RoboDK station: Proyecto_RoboDK_PR2 1.rdk

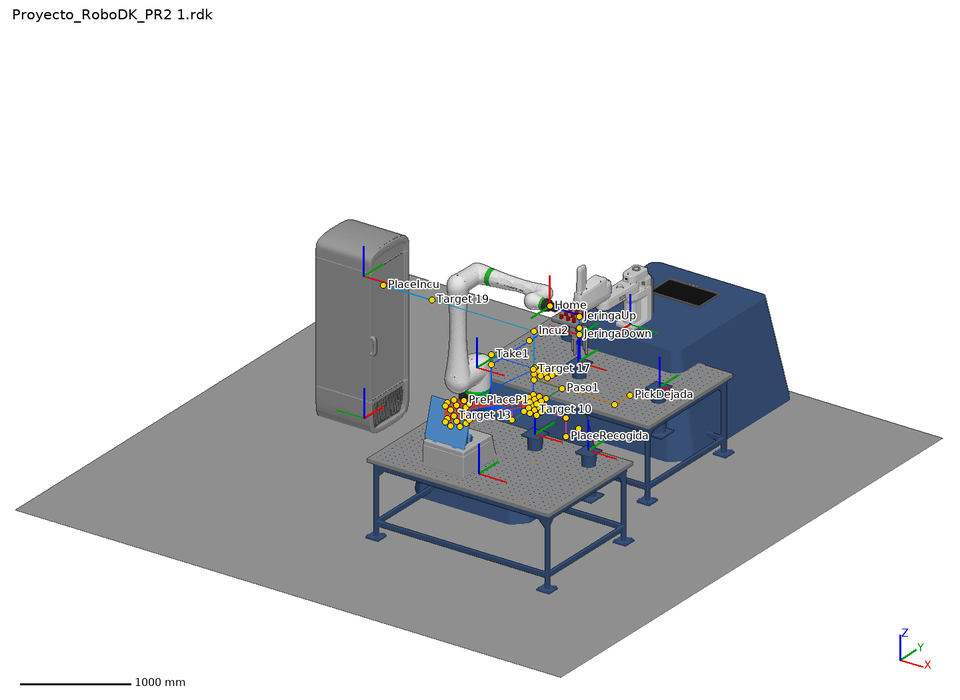
[picture v0: the station drawn from its stored meshes, robots at their saved joint values, targets as dots, program paths as lines]
Station pRUEBA (saved by RoboDK 5.9.4). Poses are relative to the parent item; angles as X-Y-Z fixed-axis rotations.
  - frame Frame 1 at (0, 0, 0) mm
    - object Floor at (-1500, 1500, 0) mm, size 3000 x 3000 x 0 mm, geometry from Floor.sld
    - object Floor at (1500, -1500, 0) mm, size 3000 x 3000 x 0 mm, geometry from Floor.sld
    - object Floor at (1500, 1500, 0) mm, size 3000 x 3000 x 0 mm, geometry from Floor.sld
    - object Floor at (-1500, -1500, 0) mm, size 3000 x 3000 x 0 mm, geometry from Floor.sld
    - object Table 2000x1200x800mm at (300, -1000, 800) mm, size 2020 x 1340 x 800 mm, geometry from Table-2000x1200x800mm.sld
    - object Table 2000x1200x800mm at (0, 1000, 800) mm, size 2020 x 1340 x 800 mm, geometry from Table-2000x1200x800mm.sld
    - object Pedestal H750mm (Type 2) at (320, 0, 0) mm, size 1266.8 x 1400.5 x 750 mm, geometry from Pedestal-H750mm-Type-2.sld
    - object Pedestal H1000mm (Type 2) at (580, 2100, 0) mm, size 1689.1 x 1867.3 x 1000 mm, geometry from Pedestal-H1000mm-Type-2.sld
    - object Pedestal H36in (Type 1) at (1400, 40, -20) mm, size 200 x 200 x 457.2 mm, geometry from Pedestal-H36in-Type-1.sld
    - object Pedestal H36in (Type 1) at (530, 40, -20) mm, size 200 x 200 x 457.2 mm, geometry from Pedestal-H36in-Type-1.sld
    - object Pedestal H36in (Type 1) at (1050, -1400, -10) mm, size 200 x 200 x 457.2 mm, geometry from Pedestal-H36in-Type-1.sld
    - object Pedestal H36in (Type 1) at (1640, -1400, -20) mm, size 200 x 200 x 457.2 mm, geometry from Pedestal-H36in-Type-1.sld
    - object Centrifugadora at (440, -1500, 800) mm, size 484.9 x 550 x 655.5 mm, geometry from Centrifugadora.stl
    - object Display Panel 24in at (590, 2390, 1010) mm, rotated rx 0 ry -90 rz 90 deg, size 43 x 556.4 x 342.2 mm, geometry from Display-Panel-24in.sld
  - frame Adept Cobra s800 Base at (530, 1620, 1000) mm, rotated rx 0 ry 0 rz -90 deg
    - robot myScara (model Adept Cobra s800): 4 axes, payload 2 kg, reach 800 mm, repeatability 0.018 mm, weight 43 kg
        modified DH rows (alpha deg, a mm, theta deg, d mm): 0, 0, 0, 0; 0, 425, 0, 0; 0, 375, 0, 184 linear; 180, 0, 0, 0
        joint limits [-105, -157.5, 0, -360] to [105, 157.5, 210, 360]; home [0, 0, 0, 0]; saved at [0, 0, 30, 90]
      - frame FrameScaraTool at (0, 0, 0) mm
        - object ScaraTool at (0, 0, 0) mm, size 193.5 x 193.5 x 277.1 mm, geometry from robodk.stl
    - target JeringaUp (Cartesian target) at (800, 0, 394) mm, rotated rx 180 ry 0 rz 0 deg; joints [0, 0, 210, 0] of myScara
    - target JeringaPreDown (Cartesian target) at (800, 0, 284) mm, rotated rx 180 ry 0 rz 0 deg; joints [0, 0, 100, 0, 0, 0] of myScara
    - target JeringaDown (Cartesian target) at (800, 0, 214) mm, rotated rx 180 ry 0 rz 0 deg; joints [0, 0, 30, 0, 0, 0] of myScara
    - target Sustancia2 (Cartesian target) at (800, 0, 214) mm, rotated rx 180 ry 0 rz -90 deg; joints [0, 0, 30, 90, 0, 0] of myScara
    - target Sustancia3 (Cartesian target) at (800, 0, 214) mm, rotated rx -180 ry 0 rz -180 deg; joints [0, 0, 30, 180, 0, 0] of myScara
    - target Alchol (Cartesian target) at (800, 0, 214) mm, rotated rx -180 ry 0 rz 90 deg; joints [0, 0, 30, 270, 0, 0] of myScara
    - target PreSustancia2 (Cartesian target) at (800, 0, 284) mm, rotated rx 180 ry 0 rz -90 deg; joints [0, 0, 100, 90] of myScara
    - target PreSustancia3 (Cartesian target) at (800, 0, 284) mm, rotated rx -180 ry 0 rz -180 deg; joints [0, 0, 100, 180] of myScara
    - target PreAlchol (Cartesian target) at (800, 0, 284) mm, rotated rx -180 ry 0 rz 90 deg; joints [0, 0, 100, 270] of myScara
    - target Target 10 (Cartesian target) at (2240, 517.5, 180) mm, rotated rx 180 ry 0 rz 90 deg; joints [143.001, -36.832, -136.065, 0, 46.065, -143.001] of myRobotUR
    - target Target 11 (Cartesian target) at (2170, 517.5, 180) mm, rotated rx 180 ry 0 rz 90 deg; joints [145.986, -35.485, -134.651, 0, 44.651, -145.986] of myRobotUR
    - target Target 12 (Cartesian target) at (2170, 590, 180) mm, rotated rx -180 ry 0 rz 90 deg; joints [148.02, -38.44, -137.769, 0, 47.769, -148.02] of myRobotUR
    - target Target 13 (Cartesian target) at (2840, 50, 230) mm, rotated rx 180 ry 0 rz 90 deg; joints [106.738, -40.272, -144.565, 0, 54.565, -106.738] of myRobotUR
    - target Target 14 (Cartesian target) at (2240, 590, 180) mm, rotated rx -180 ry 0 rz 90 deg; joints [145.135, -39.762, -139.179, 0, 49.179, -145.135] of myRobotUR
    - target Target 15 (Cartesian target) at (2315, 590, 180) mm, rotated rx 180 ry 0 rz 90 deg; joints [142.232, -41.383, -140.921, 0, 50.921, -142.232] of myRobotUR
    - target Target 16 (Cartesian target) at (2315, 590, 180) mm, rotated rx 180 ry 0 rz 90 deg; joints [142.232, -41.383, -140.921, 0, 50.921, -142.232] of myRobotUR
    - target Target 17 (Cartesian target) at (2170, 450, 540) mm, rotated rx 180 ry 0 rz 90 deg; joints [143.864, -20.056, -157.055, 0, 67.055, -143.864] of myRobotUR
    - target Target 18 (Cartesian target) at (1795, 200, -45) mm, rotated rx 0 ry -90 rz -90 deg; joints [12.327, 57.498, -112.698, -13.327, 112.147, -5.103] of myRobotUR
    - target Target 19 (Cartesian target) at (1355, -1230, 440) mm, rotated rx 0 ry -90 rz 90 deg; joints [162.189, 12.692, -58.671, 20.612, 60.328, -10.547] of myRobotUR
    - target Target 20 (Cartesian target) at (2140, 200, -50) mm, rotated rx 0 ry -90 rz -90 deg; joints [-25.299, 52.835, -105.784, 26.16, 104.237, 6.888] of myRobotUR
    - target Target 21 (Cartesian target) at (1120, -100, -45) mm, rotated rx 0 ry -90 rz 0 deg; joints [64.725, 54.326, -114.186, 27.366, 111.745, 10.855] of myRobotUR
    - target Target 22 (Cartesian target) at (800, 0, 214) mm, rotated rx 180 ry 0 rz 0 deg; joints [72.717, 31.504, -45.613, 0, -44.387, -162.717] of myRobotUR
    - target Target 23 (Cartesian target) at (1905, 450, 1070) mm, rotated rx 0 ry -90 rz -90 deg; joints [0, 0, 0, 0, 0, 0] of myRobotUR
  - frame Fanuc CRX-25iA Base at (50, -100, 1120) mm
    - robot myRobotUR (model Fanuc CRX-25iA): 6 axes, payload 25 kg, reach 1889 mm, repeatability 0.05 mm, weight 135 kg
        modified DH rows (alpha deg, a mm, theta deg, d mm): 0, 0, 0, 370; -90, 0, -90, 0; 0, 950, 0, 0; -90, 0, 0, 750; 90, 0, 0, -185; -90, 0, 0, 180
        base shift (0, 0, -370) mm
        joint limits [-180, -180, -270, -190, -180, -225] to [180, 180, 270, 190, 180, 225]; home [0, 0, 0, 0, 0, 0]; saved at [0, 0, 0, 0, 0, 0]
      - frame RobotiQ 2F-140 Gripper (Mechanism) Base at (0, 0, 0) mm
        - robot RobotiQ 2F-140 Gripper (Mechanism) (model RobotiQ 2F140): 1 axes, payload 5 kg
            joint limits [0] to [140]; home [140]; saved at [40]
          - tool Tool 1, TCP at (0, 0, 200) mm
            - object Soporte1 at (-20, 30, 45) mm, rotated rx 90 ry 0 rz 90 deg, size 266.4 x 266.4 x 36 mm, geometry from soporteprobeta.stl
              - object P1 at (5, 0, 0) mm, size 36.4 x 36.5 x 72.9 mm, geometry from probeta.stl
              - object P2 at (75, 0, 0) mm, size 36.4 x 36.5 x 72.9 mm, geometry from probeta.stl
              - object P3 at (150, 0, 0) mm, size 36.4 x 36.5 x 72.9 mm, geometry from probeta.stl
              - object P4 at (150, 72.5, 0) mm, size 36.4 x 36.5 x 72.9 mm, geometry from probeta.stl
              - object P5 at (75, 72.5, 0) mm, size 36.4 x 36.5 x 72.9 mm, geometry from probeta.stl
              - object P6 at (5, 72.5, 0) mm, size 36.4 x 36.5 x 72.9 mm, geometry from probeta.stl
              - object P7 at (5, 145, 0) mm, size 36.4 x 36.5 x 72.9 mm, geometry from probeta.stl
              - object P8 at (75, 145, 0) mm, size 36.4 x 36.5 x 72.9 mm, geometry from probeta.stl
              - object P9 at (150, 145, 0) mm, size 36.4 x 36.5 x 72.9 mm, geometry from probeta.stl
        - target GarraOpen (Cartesian target) at (0, 0, 0) mm; joints [140, 0, 0, 0, 0, 0] of RobotiQ 2F-140 Gripper (Mechanism)
        - target GarraPick (Cartesian target) at (0, 0, 0) mm; joints [40, 0, 30, 270] of RobotiQ 2F-140 Gripper (Mechanism)
  - frame IncubadoraMECA at (-1500, 340, 0) mm, rotated rx 0 ry 0 rz 90 deg
    - robot Refrigeradora: 1 axes
        modified DH rows (alpha deg, a mm, theta deg, d mm): 0, 0, 0, 0 linear
        base shift (0, 0, 0) mm, rotated rx 0 ry 90 rz 0 deg
        joint limits [0] to [600]; home [0]; saved at [0]
    - target DoorClose (Cartesian target) at (0, 0, 0) mm; joints [0, 54.489, -114.295, 25.89, 112.102, 10.349] of Refrigeradora
    - target DoorOpen (Cartesian target) at (600, 0, 0) mm; joints [600, 54.489, -114.295, 25.89, 112.102, 10.349] of Refrigeradora
  - frame Dejada at (1410, 820, 940) mm
    - target PickDejada (Cartesian target) at (-100, -315, 15) mm, rotated rx 0 ry -90 rz -90 deg; joints [21.278, 62.791, -64.214, 70.676, 80.917, -24.237] of myRobotUR
    - target PrePickDejada (Cartesian target) at (-100, -555, 15) mm, rotated rx 0 ry -90 rz -90 deg; joints [9.654, 60.648, -68.477, 81.008, 86.473, -21.245] of myRobotUR
    - target Home (Cartesian target) at (-430, -1105, 1130) mm, rotated rx 0 ry -90 rz -180 deg; joints [0, 0, 0, 0, 0, 0] of myRobotUR
  - frame Pinchazo at (520, 820, 940) mm
    - target PlacePinchazo/Pin2 (Cartesian target) at (-90, -320, 15) mm, rotated rx 0 ry -90 rz -90 deg; joints [64.725, 54.326, -114.186, 27.366, 111.745, 10.855] of myRobotUR
    - target PrePlacePinchazo (Cartesian target) at (-100, -555, 15) mm, rotated rx 0 ry -90 rz -90 deg; joints [39.607, 59.804, -135.062, 59.694, 116.826, 37.672] of myRobotUR
    - target Pin1 (Cartesian target) at (-20, -320, 15) mm, rotated rx 0 ry -90 rz -90 deg; joints [57.411, 52.743, -110.092, 34.243, 106.825, 11.146] of myRobotUR
    - target Pin3 (Cartesian target) at (-170, -320, 15) mm, rotated rx 0 ry -90 rz -90 deg; joints [74.441, 56.789, -118.585, 17.593, 117.447, 8.315] of myRobotUR
    - target Pin4 (Cartesian target) at (-170, -390, 15) mm, rotated rx 0 ry -90 rz -90 deg; joints [71.034, 59.762, -126.932, 23.265, 124.628, 13.729] of myRobotUR
    - target Pin5 (Cartesian target) at (-90, -390, 15) mm, rotated rx 0 ry -90 rz -90 deg; joints [59.932, 55.868, -120.613, 33.929, 116.149, 16.513] of myRobotUR
    - target Pin6 (Cartesian target) at (-20, -390, 15) mm, rotated rx 0 ry -90 rz -90 deg; joints [52.114, 53.534, -115.301, 40.717, 109.712, 16.188] of myRobotUR
    - target Pin7 (Cartesian target) at (-20, -460, 15) mm, rotated rx 0 ry -90 rz -90 deg; joints [45.12, 54.354, -120.163, 49.035, 110.857, 22.297] of myRobotUR
    - target Pin8 (Cartesian target) at (-90, -460, 15) mm, rotated rx 0 ry -90 rz -90 deg; joints [52.947, 57.441, -126.856, 43.337, 118.6, 24.308] of myRobotUR
    - target Pin9 (Cartesian target) at (-170, -460, 15) mm, rotated rx 0 ry -90 rz -90 deg; joints [65.053, 62.974, -135.774, 33.701, 130.522, 23.429] of myRobotUR
  - frame Incubadora at (-1500, 330, 1430) mm
    - target EncaraIncu (Cartesian target) at (1920, -65, -475) mm, rotated rx 0 ry -90 rz 0 deg; joints [18.17, 52.517, -103.492, 161.349, 77.192, 4.279] of myRobotUR
    - target Incu2 (Cartesian target) at (1920, -65, 10) mm, rotated rx 0 ry -90 rz 0 deg; joints [18.423, 11.864, -59.167, 158.797, 119.096, -10.683] of myRobotUR
    - target PlaceIncu (Cartesian target) at (260, -65, 10) mm, rotated rx 0 ry -90 rz 0 deg; joints [170.623, 35.683, -40.43, 14.285, 41.321, -10.826] of myRobotUR
    - target PrePlaceIncu (Cartesian target) at (800, -65, 10) mm, rotated rx 0 ry -90 rz 0 deg; joints [162.189, 12.692, -58.671, 20.612, 60.328, -10.547] of myRobotUR
  - frame Centrifugadora at (1050, -620, 940) mm
    - target Centri1 (Cartesian target) at (-550, 885, 500) mm, rotated rx 0 ry -90 rz 0 deg; joints [16.192, 15.174, -57.101, 160.923, 121.44, -10.226] of myRobotUR
    - target Centri2 (Cartesian target) at (-550, 700, 500) mm, rotated rx 0 ry -90 rz 0 deg; joints [-0.454, 11.696, -54.321, 180.559, 125.678, 0.326] of myRobotUR
    - target Centri3/Giro (Cartesian target) at (-550, 700, 500) mm, rotated rx 0 ry -90 rz -90 deg; joints [0, 0.179, -68.498, 90, 90, -21.502] of myRobotUR
    - target Centri4/Giro (Cartesian target) at (-550, 700, 500) mm, rotated rx 0 ry -90 rz -180 deg; joints [49.88, -8.528, -41.712, -60.721, 61.247, 40.627] of myRobotUR
    - target Centri5 (Cartesian target) at (-550, 100, 500) mm, rotated rx 0 ry -90 rz -180 deg; joints [-41.992, 3.157, -65.505, 44.688, 72.052, -16.952] of myRobotUR
    - target PrePlaceCentri (Cartesian target) at (-550, 100, 10) mm, rotated rx 0 ry -90 rz -180 deg; joints [136.977, -56.167, -55.961, -131.602, 114.156, 24.744] of myRobotUR
    - target PlaceCentri (Cartesian target) at (-320, 100, 10) mm, rotated rx 0 ry -90 rz -180 deg; joints [154.701, -52.835, -74.216, -153.84, 104.237, 6.888] of myRobotUR
    - target LlevarRecogida (Cartesian target) at (-320, 100, 200) mm, rotated rx 0 ry -90 rz -180 deg; joints [154.826, -35.816, -89.736, -154.826, 90.239, 0.112] of myRobotUR
    - target Paso1 (Cartesian target) at (-320, 885, 15) mm, rotated rx 0 ry -90 rz -90 deg; joints [20.272, 50.493, -105.389, 70.399, 95.275, 14.477] of myRobotUR
    - target Paso2 (Cartesian target) at (-320, 885, 15) mm, rotated rx 0 ry -90 rz -180 deg; joints [47.726, 52.078, -90.466, -47.727, 90.314, -0.345] of myRobotUR
    - target PrePaso3 (Cartesian target) at (-320, 445, 15) mm, rotated rx 0 ry -90 rz 180 deg; joints [12.327, 57.498, -112.698, -13.327, 112.147, -5.103] of myRobotUR
    - target Take1 (Cartesian target) at (-550, 100, 600) mm, rotated rx 0 ry -90 rz -180 deg; joints [136.75, 4.022, -125.669, -130.814, 64.868, -26.187] of myRobotUR
    - target Take2 (Cartesian target) at (-550, 100, 600) mm, rotated rx 180 ry 0 rz 0 deg; joints [119.485, 4.704, -152.458, 0, 62.458, -119.485] of myRobotUR
    - target Take3 (Cartesian target) at (-70, 100, 600) mm, rotated rx 180 ry 0 rz 0 deg; joints [145.25, -19.338, -156.721, 0, 66.721, -145.25] of myRobotUR
    - target Take4 (Cartesian target) at (-70, 70, 600) mm, rotated rx -180 ry 0 rz 0 deg; joints [143.864, -20.056, -157.055, 0, 67.055, -143.864] of myRobotUR
    - target PickP1 (Cartesian target) at (-70, 70, 240) mm, rotated rx 180 ry 0 rz 0 deg; joints [143.864, -32.854, -131.921, 0, 41.921, -143.864] of myRobotUR
    - target PrePickP1 (Cartesian target) at (-70, 70, 350) mm, rotated rx 180 ry 0 rz 0 deg; joints [143.864, -28.076, -139.387, 0, 49.387, -143.864] of myRobotUR
    - target PickP2 (Cartesian target) at (-70, 0, 240) mm, rotated rx 180 ry 0 rz 0 deg; joints [140.79, -34.237, -133.35, 0, 43.35, -140.79] of myRobotUR
    - target PrePickP2 (Cartesian target) at (-70, 0, 350) mm, rotated rx 180 ry 0 rz 0 deg; joints [140.79, -29.624, -140.622, 0, 50.622, -140.79] of myRobotUR
    - target PickP3 (Cartesian target) at (-70, -75, 240) mm, rotated rx -180 ry 0 rz 0 deg; joints [137.743, -35.912, -135.097, 0, 45.097, -137.743] of myRobotUR
    - target PrePickP3 (Cartesian target) at (-70, -75, 350) mm, rotated rx -180 ry 0 rz 0 deg; joints [137.743, -31.486, -142.156, 0, 52.156, -137.743] of myRobotUR
    - target PickP4 (Cartesian target) at (-2.5, -75, 240) mm, rotated rx -180 ry 0 rz 0 deg; joints [140.019, -38.472, -137.802, 0, 47.802, -140.019] of myRobotUR
    - target PrePickP4 (Cartesian target) at (-2.5, -75, 350) mm, rotated rx -180 ry 0 rz 0 deg; joints [140.019, -34.309, -144.577, 0, 54.577, -140.019] of myRobotUR
    - target PickP5 (Cartesian target) at (-2.5, 0, 240) mm, rotated rx 180 ry 0 rz 0 deg; joints [143.001, -36.832, -136.065, 0, 46.065, -143.001] of myRobotUR
    - target PrePickP5 (Cartesian target) at (-2.5, 0, 350) mm, rotated rx 180 ry 0 rz 0 deg; joints [143.001, -32.503, -143.016, 0, 53.016, -143.001] of myRobotUR
    - target PickP6 (Cartesian target) at (-2.5, 70, 240) mm, rotated rx 180 ry 0 rz 0 deg; joints [145.986, -35.485, -134.651, 0, 44.651, -145.986] of myRobotUR
    - target PrePickP6 (Cartesian target) at (-2.5, 70, 350) mm, rotated rx -180 ry 0 rz 0 deg; joints [145.986, -31.013, -141.762, 0, 51.762, -145.986] of myRobotUR
    - target PickP7 (Cartesian target) at (70, 70, 240) mm, rotated rx 180 ry 0 rz 0 deg; joints [148.02, -38.44, -137.769, 0, 47.769, -148.02] of myRobotUR
    - target PrePickP7 (Cartesian target) at (70, 70, 350) mm, rotated rx 180 ry 0 rz 0 deg; joints [148.02, -34.274, -144.546, 0, 54.546, -148.02] of myRobotUR
    - target PickP8 (Cartesian target) at (70, 0, 240) mm, rotated rx 180 ry 0 rz 0 deg; joints [145.135, -39.762, -139.179, 0, 49.179, -145.135] of myRobotUR
    - target PrePickP8 (Cartesian target) at (70, 0, 350) mm, rotated rx -180 ry 0 rz 0 deg; joints [145.135, -35.723, -145.828, 0, 55.828, -145.135] of myRobotUR
    - target PickP9 (Cartesian target) at (70, -75, 240) mm, rotated rx 180 ry 0 rz 0 deg; joints [142.232, -41.383, -140.921, 0, 50.921, -142.232] of myRobotUR
    - target PrePickP9 (Cartesian target) at (70, -75, 350) mm, rotated rx -180 ry 0 rz 0 deg; joints [142.232, -37.492, -147.428, 0, 57.428, -142.232] of myRobotUR
    - target PlaceP1 (Cartesian target) at (-390, -560, 290) mm, rotated rx -180 ry 0 rz 0 deg; joints [110.881, -40.337, -144.63, 0, 54.63, -110.881] of myRobotUR
    - target PrePlaceP1 (Cartesian target) at (-390, -560, 450) mm, rotated rx -180 ry 0 rz 0 deg; joints [110.881, -35.397, -154.371, 0, 64.371, -110.881] of myRobotUR
    - target PlaceP2 (Cartesian target) at (-290, -665, 290) mm, rotated rx 180 ry 0 rz 0 deg; joints [113.232, -47.852, -152.398, 0, 62.398, -113.232] of myRobotUR
    - target PrePlaceP2 (Cartesian target) at (-290, -665, 450) mm, rotated rx -180 ry 0 rz 0 deg; joints [113.232, -43.764, -161.652, 0, 71.652, -113.232] of myRobotUR
    - target PlaceP3 (Cartesian target) at (-380, -780, 290) mm, rotated rx -180 ry 0 rz 0 deg; joints [108.118, -51.381, -156.177, 0, 66.177, -108.118] of myRobotUR
    - target PrePlace3 (Cartesian target) at (-380, -780, 450) mm, rotated rx 180 ry 0 rz 0 deg; joints [108.118, -47.7, -165.375, 0, 75.375, -108.118] of myRobotUR
    - target PlaceP4 (Cartesian target) at (-490, -675, 290) mm, rotated rx 180 ry 0 rz 0 deg; joints [104.926, -43.35, -147.695, 0, 57.695, -104.926] of myRobotUR
    - target PrePlace4 (Cartesian target) at (-490, -675, 450) mm, rotated rx 180 ry 0 rz 0 deg; joints [104.926, -38.757, -157.185, 0, 67.185, -104.926] of myRobotUR
    - target PlaceP5 (Cartesian target) at (-310, -590, 290) mm, rotated rx -180 ry 0 rz 0 deg; joints [113.729, -43.755, -148.113, 0, 58.113, -113.729] of myRobotUR
    - target PrePlace5 (Cartesian target) at (-310, -590, 450) mm, rotated rx -180 ry 0 rz 0 deg; joints [113.729, -39.209, -157.575, 0, 67.575, -113.729] of myRobotUR
    - target PlaceP6 (Cartesian target) at (-300, -750, 290) mm, rotated rx -180 ry 0 rz 0 deg; joints [111.533, -52.005, -156.854, 0, 66.854, -111.533] of myRobotUR
    - target PrePlace6 (Cartesian target) at (-300, -750, 450) mm, rotated rx 180 ry 0 rz 0 deg; joints [111.533, -48.399, -166.055, 0, 76.055, -111.533] of myRobotUR
    - target PlaceP7 (Cartesian target) at (-460, -750, 290) mm, rotated rx -180 ry 0 rz 0 deg; joints [105.331, -47.772, -152.313, 0, 62.313, -105.331] of myRobotUR
    - target PrePlace7 (Cartesian target) at (-460, -750, 450) mm, rotated rx -180 ry 0 rz 0 deg; joints [105.331, -43.675, -161.571, 0, 71.571, -105.331] of myRobotUR
    - target PlaceP8 (Cartesian target) at (-470, -600, 290) mm, rotated rx 180 ry 0 rz 0 deg; joints [106.738, -40.272, -144.565, 0, 54.565, -106.738] of myRobotUR
    - target PrePlace8 (Cartesian target) at (-470, -600, 450) mm, rotated rx -180 ry 0 rz 0 deg; joints [106.738, -35.325, -154.313, 0, 64.313, -106.738] of myRobotUR
    - target PlaceP9 (Cartesian target) at (-390, -670, 290) mm, rotated rx -180 ry 0 rz 0 deg; joints [109.188, -45.379, -149.798, 0, 59.798, -109.188] of myRobotUR
    - target PrePlaceP9 (Cartesian target) at (-390, -670, 450) mm, rotated rx -180 ry 0 rz 0 deg; joints [109.188, -41.015, -159.161, 0, 69.161, -109.188] of myRobotUR
  - frame Recogida at (1640, -620, 940) mm
    - target PlaceRecogida (Cartesian target) at (-320, 100, 10) mm, rotated rx 0 ry -90 rz 180 deg; joints [-12.208, 58.427, -65.934, 13.33, 66.511, -5.395] of myRobotUR
    - target PrePlaceRecogdia (Cartesian target) at (-320, 100, 200) mm, rotated rx 0 ry -90 rz 180 deg; joints [-12.25, 48.617, -57.534, 14.432, 58.36, -7.688] of myRobotUR
    - target Retirada (Cartesian target) at (-320, 300, 10) mm, rotated rx 0 ry -90 rz 180 deg; joints [-1.84, 56.994, -66.931, 2, 66.943, -0.783] of myRobotUR
  - program HomeRobot (2 instructions, listed below)
  - program ResetSoporte (1 instructions, listed below)
  - program AbrirGarra (2 instructions, listed below)
  - program CerrarGarra (2 instructions, listed below)
  - program SubirJeringa (5 instructions, listed below)
  - program BajarJeringa (5 instructions, listed below)
  - program DoorClose (2 instructions, listed below)
  - program DoorOpen (2 instructions, listed below)
  - program Probetas (2 instructions, listed below)
  - program ResetProbetas (9 instructions, listed below)
  - Python program OcultarProbetas (listed below)
  - Python program MostrarProbetas (listed below)
  - program Adjuntar Soporte (1 instructions, listed below)
  - program PincharAlchol (4 instructions, listed below)
  - program Pinchar3Sustancias (8 instructions, listed below)
  - program DeDejadaAPinchazo (8 instructions, listed below)
  - program DePinchazoAIncu (9 instructions, listed below)
  - program DeIncuACentri (9 instructions, listed below)
  - program DeCentriAPinchazo (9 instructions, listed below)
  - program DePinchazoACentri (9 instructions, listed below)
  - program DeCentriARecogida (9 instructions, listed below)
  - program ProgramaSustancias (21 instructions, listed below)
  - program PrgramaAlchol (20 instructions, listed below)
  - program MeterProbetas (72 instructions, listed below)
  - program SacarProbetas (74 instructions, listed below)
  - program ProgramaUniversal (5 instructions, listed below)
  - program PincharSustancia1 (3 instructions, listed below)
  - program PincharSustancia2 (3 instructions, listed below)
  - program PincharSustancia3 (4 instructions, listed below)
  - Python program MqttListener (listed below)
  - Python program PresenciaSoporte (listed below)
  - Python program RobotController (listed below)
  - Python program ScaraController (listed below)
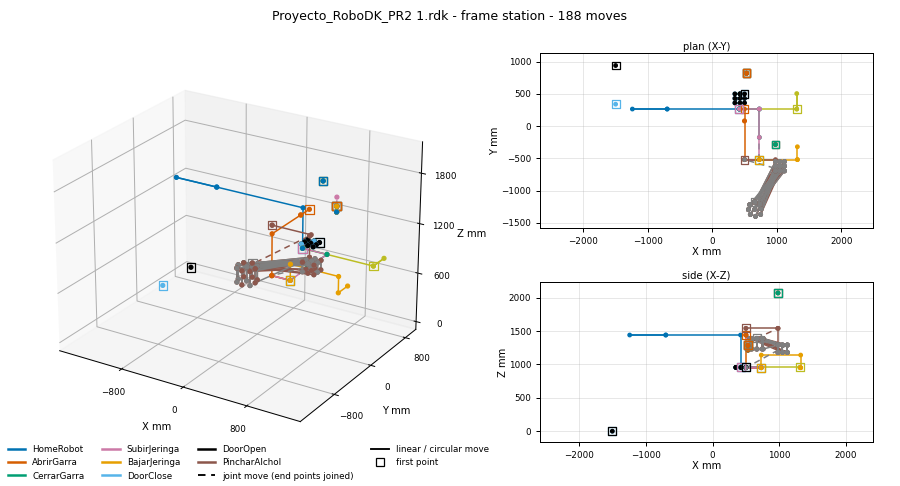
[picture p0: tool path of Proyecto_RoboDK_PR2 1.rdk in frame station, 188 of 188 moves have a stored position in this frame; points joined in program order, loops and branches not executed]

--- program HomeRobot (robot myRobotUR) ---
  Est. Ref.: Dejada
  MoveJ (Home)

--- program ResetSoporte (robot myRobotUR) ---
  Reemplazar Soporte1

--- program AbrirGarra (robot RobotiQ 2F-140 Gripper (Mechanism)) ---
  Set Ref.: RobotiQ 2F-140 Gripper (Mechanism) Base
  MoveJ (GarraOpen)

--- program CerrarGarra (robot RobotiQ 2F-140 Gripper (Mechanism)) ---
  Set Ref.: RobotiQ 2F-140 Gripper (Mechanism) Base
  MoveJ (GarraPick)

--- program SubirJeringa (robot myScara) ---
  Set Ref.: Adept Cobra s800 Base
  Set speed (50.0 mm/s)
  MoveJ (JeringaPreDown)
  Set speed (100.0 mm/s)
  MoveJ (JeringaUp)

--- program BajarJeringa (robot myScara) ---
  Set Ref.: Adept Cobra s800 Base
  Set speed (500.0 mm/s)
  MoveJ (JeringaPreDown)
  Set speed (500.0 mm/s)
  MoveJ (JeringaDown)

--- program DoorClose (robot Refrigeradora) ---
  Est. Ref.: IncubadoraMECA
  MoveJ (DoorClose)

--- program DoorOpen (robot Refrigeradora) ---
  Est. Ref.: IncubadoraMECA
  MoveJ (DoorOpen)

--- program Probetas (robot myRobotUR) ---
  Adjuntar a Tool 1
  Separar de Tool 1

--- program ResetProbetas (robot myRobotUR) ---
  Reemplazar P1
  Reemplazar P2
  Reemplazar P3
  Reemplazar P4
  Reemplazar P5
  Reemplazar P6
  Reemplazar P7
  Reemplazar P8
  Reemplazar P9

--- Python program OcultarProbetas ---
# Type help("robodk.robolink") or help("robodk.robomath") for more information
# Press F5 to run the script
# Documentation: https://robodk.com/doc/en/RoboDK-API.html
# Reference:     https://robodk.com/doc/en/PythonAPI/robodk.html
# Note: It is not required to keep a copy of this file, your Python script is saved with your RDK project

from robodk import robolink
from robodk import robomath

RDK = robolink.Robolink()

NUM_SOPORTES = 4


for i in range(1, NUM_SOPORTES + 1):
    soporte = RDK.Item(f"Soporte{i}", robolink.ITEM_TYPE_OBJECT)

    if soporte.Valid():
        # Ocultar soporte
        soporte.setVisible(False)

        # Obtener TODOS los hijos del soporte (las probetas)
        hijos = soporte.Childs()

        for probeta in hijos:
            probeta.setVisible(False)

--- Python program MostrarProbetas ---
# Type help("robodk.robolink") or help("robodk.robomath") for more information
# Press F5 to run the script
# Documentation: https://robodk.com/doc/en/RoboDK-API.html
# Reference:     https://robodk.com/doc/en/PythonAPI/robodk.html
# Note: It is not required to keep a copy of this file, your Python script is saved with your RDK project

from robodk import robolink
from robodk import robomath

RDK = robolink.Robolink()

NUM_SOPORTES = 4

for i in range(1, NUM_SOPORTES + 1):
    soporte = RDK.Item(f"Soporte{i}", robolink.ITEM_TYPE_OBJECT)

    if soporte.Valid():
        # Ocultar soporte
        soporte.setVisible(True)

        # Obtener TODOS los hijos del soporte (las probetas)
        hijos = soporte.Childs()

        for probeta in hijos:
            probeta.setVisible(True)

--- program Adjuntar Soporte (robot myRobotUR) ---
  Adjuntar a Tool 1

--- program PincharAlchol (robot myScara) ---
  Est. Ref.: Adept Cobra s800 Base
  MoveJ (PreAlchol)
  MoveJ (Alchol)
  MoveJ (PreAlchol)

--- program Pinchar3Sustancias (robot myScara) ---
  Est. Ref.: Adept Cobra s800 Base
  MoveJ (JeringaPreDown)
  MoveJ (JeringaDown)
  MoveJ (PreSustancia2)
  MoveJ (Sustancia2)
  MoveJ (PreSustancia3)
  MoveJ (Sustancia3)
  MoveJ (JeringaPreDown)

--- program DeDejadaAPinchazo (robot myRobotUR) ---
  Est. Ref.: Dejada
  MoveJ (PrePickDejada)
  MoveL (PickDejada)
  Adjuntar a Tool 1
  MoveL (PrePickDejada)
  Est. Ref.: Pinchazo
  MoveL (PrePlacePinchazo)
  MoveL (PlacePinchazo) -> target PlacePinchazo/Pin2

--- program DePinchazoAIncu (robot myRobotUR) ---
  Est. Ref.: Pinchazo
  MoveL (PrePlacePinchazo)
  Est. Ref.: Incubadora
  MoveJ (EncaraIncu)
  MoveL (Incu2)
  MoveL (PrePlaceIncu)
  MoveL (PlaceIncu)
  Separar de Tool 1
  MoveL (PrePlaceIncu)

--- program DeIncuACentri (robot myRobotUR) ---
  Est. Ref.: Centrifugadora
  MoveL (Centri1)
  MoveL (Centri2)
  MoveL (Centri3/Giro)
  MoveL (Centri5)
  MoveL (PrePlaceCentri)
  MoveL (PlaceCentri)
  Separar de Tool 1
  MoveL (PrePlaceCentri)

--- program DeCentriAPinchazo (robot myRobotUR) ---
  Est. Ref.: Centrifugadora
  MoveL (PlaceCentri)
  Adjuntar a Tool 1
  MoveJ (PrePaso3)
  MoveL (Paso2)
  MoveL (Paso1)
  Est. Ref.: Pinchazo
  MoveL (PrePlacePinchazo)
  MoveL (PlacePinchazo) -> target PlacePinchazo/Pin2

--- program DePinchazoACentri (robot myRobotUR) ---
  Est. Ref.: Pinchazo
  MoveL (PrePlacePinchazo)
  Est. Ref.: Centrifugadora
  MoveL (Paso1)
  MoveL (Paso2)
  MoveL (PrePaso3)
  MoveL (PlaceCentri)
  Separar de Tool 1
  MoveL (PrePlaceCentri)

--- program DeCentriARecogida (robot myRobotUR) ---
  Est. Ref.: Centrifugadora
  MoveL (PlaceCentri)
  Adjuntar a Tool 1
  MoveL (Recogida1) -> target LlevarRecogida
  Est. Ref.: Recogida
  MoveL (PrePlaceRecogdia)
  MoveL (PlaceRecogida)
  Separar de Tool 1
  MoveL (Retirada)

--- program ProgramaSustancias (robot myRobotUR) ---
  Est. Ref.: Pinchazo
  MoveL (Pin1)
  Llamar Program1
  Llamar Pinchar3Sustancias
  MoveL (PlacePinchazo/Pin2)
  Llamar Pinchar3Sustancias
  MoveL (Pin3)
  Llamar Pinchar3Sustancias
  MoveL (Pin4)
  Llamar Pinchar3Sustancias
  MoveL (Pin5)
  Llamar Pinchar3Sustancias
  MoveL (Pin6)
  Llamar Pinchar3Sustancias
  MoveL (Pin7)
  Llamar Pinchar3Sustancias
  MoveL (Pin8)
  Llamar Pinchar3Sustancias
  MoveL (Pin9)
  Llamar Pinchar3Sustancias
  MoveJ (PlacePinchazo/Pin2)

--- program PrgramaAlchol (robot myRobotUR) ---
  Est. Ref.: Pinchazo
  MoveL (Pin1)
  Llamar PincharAlchol
  MoveL (PlacePinchazo/Pin2)
  Llamar PincharAlchol
  MoveL (Pin3)
  Llamar PincharAlchol
  MoveL (Pin4)
  Llamar PincharAlchol
  MoveL (Pin5)
  Llamar PincharAlchol
  MoveL (Pin6)
  Llamar PincharAlchol
  MoveL (Pin7)
  Llamar PincharAlchol
  MoveL (Pin8)
  Llamar PincharAlchol
  MoveL (Pin9)
  Llamar PincharAlchol
  MoveJ (PlacePinchazo/Pin2)

--- program MeterProbetas (robot myRobotUR) ---
  Est. Ref.: Centrifugadora
  MoveJ (Take1)
  MoveL (Take2)
  MoveL (Take3)
  MoveL (Take4)
  MoveL (PrePickP1)
  MoveL (PickP1)
  Adjuntar a Tool 1
  MoveL (PrePickP1)
  MoveL (PrePlaceP1)
  MoveL (PlaceP1)
  Separar de Tool 1
  MoveL (PrePlaceP1)
  MoveL (PrePickP2)
  MoveL (PickP2)
  Adjuntar a Tool 1
  MoveL (PrePickP2)
  MoveL (PrePlaceP2)
  MoveL (PlaceP2)
  Separar de Tool 1
  MoveL (PrePlaceP2)
  MoveL (PrePickP3)
  MoveL (PickP3)
  Adjuntar a Tool 1
  MoveL (PrePickP3)
  MoveL (PrePlace3)
  MoveL (PlaceP3)
  Separar de Tool 1
  MoveL (PrePlace3)
  MoveL (PrePickP4)
  MoveL (PickP4)
  Adjuntar a Tool 1
  MoveL (PrePlace4)
  MoveL (PlaceP4)
  Separar de Tool 1
  MoveL (PrePlace4)
  MoveL (PrePickP5)
  MoveL (PickP5)
  Adjuntar a Tool 1
  MoveL (PrePlace5)
  MoveL (PlaceP5)
  Separar de Tool 1
  MoveL (PrePlace5)
  MoveL (PrePickP6)
  MoveL (PickP6)
  Adjuntar a Tool 1
  MoveL (PrePlace6)
  MoveL (PlaceP6)
  Separar de Tool 1
  MoveL (PrePlace6)
  MoveL (PrePickP7)
  MoveL (PickP7)
  Adjuntar a Tool 1
  MoveL (PrePlace7)
  MoveL (PlaceP7)
  Separar de Tool 1
  MoveL (PrePlace7)
  MoveL (PrePickP8)
  MoveL (PickP8)
  Adjuntar a Tool 1
  MoveL (PrePlace8)
  MoveL (PlaceP8)
  Separar de Tool 1
  MoveL (PrePlace8)
  MoveL (PrePickP9)
  MoveL (PickP9)
  Adjuntar a Tool 1
  MoveL (PrePlaceP9)
  MoveL (PlaceP9)
  Separar de Tool 1
  MoveL (PrePlaceP9)
  MoveJ (Take4)

--- program SacarProbetas (robot myRobotUR) ---
  Est. Ref.: Centrifugadora
  MoveL (PrePlaceP1)
  MoveL (PlaceP1)
  Adjuntar a Tool 1
  MoveJ (PrePlaceP1)
  MoveL (PrePickP1)
  MoveL (PickP1)
  Separar de Tool 1
  MoveL (PrePickP1)
  MoveJ (PrePlaceP2)
  MoveL (PlaceP2)
  Adjuntar a Tool 1
  MoveL (PrePickP2)
  MoveL (PickP2)
  Separar de Tool 1
  MoveL (PrePickP2)
  MoveJ (PrePlace3)
  MoveL (PlaceP3)
  Adjuntar a Tool 1
  MoveL (PrePlace3)
  MoveL (PrePickP3)
  MoveL (PickP3)
  Separar de Tool 1
  MoveL (PrePickP3)
  MoveL (PrePlace4)
  MoveJ (PlaceP4)
  Adjuntar a Tool 1
  MoveL (PrePlace4)
  MoveL (PrePickP4)
  MoveL (PickP4)
  Separar de Tool 1
  MoveL (PrePickP4)
  MoveL (PrePlace5)
  MoveJ (PlaceP5)
  Adjuntar a Tool 1
  MoveL (PrePlace5)
  MoveL (PrePickP5)
  MoveL (PickP5)
  Separar de Tool 1
  MoveL (PrePickP5)
  MoveL (PrePlace6)
  MoveJ (PlaceP6)
  Adjuntar a Tool 1
  MoveL (PrePlace6)
  MoveL (PrePickP6)
  MoveL (PickP6)
  Separar de Tool 1
  MoveL (PrePickP6)
  MoveL (PrePlace7)
  MoveJ (PlaceP7)
  Adjuntar a Tool 1
  MoveL (PrePlace7)
  MoveL (PrePickP7)
  MoveL (PickP7)
  Separar de Tool 1
  MoveL (PrePickP7)
  MoveL (PrePlace8)
  MoveJ (PlaceP8)
  Adjuntar a Tool 1
  MoveL (PrePlace8)
  MoveL (PrePickP8)
  MoveL (PickP8)
  Separar de Tool 1
  MoveL (PrePickP8)
  MoveL (PrePlaceP9)
  MoveJ (PlaceP9)
  Adjuntar a Tool 1
  MoveL (PrePlaceP9)
  MoveL (PrePickP9)
  MoveL (PickP9)
  Separar de Tool 1
  MoveL (PrePickP9)
  MoveJ (PrePlaceCentri)
  Llamar ResetProbetas

--- program ProgramaUniversal (robot myRobotUR) ---
  Llamar ScaraController
  Llamar DoorOpen
  Llamar DePinchazoAIncu
  Llamar DoorClose
  Llamar RobotController

--- program PincharSustancia1 (robot myScara) ---
  Est. Ref.: Adept Cobra s800 Base
  MoveJ (JeringaPreDown)
  MoveJ (JeringaDown)

--- program PincharSustancia2 (robot myScara) ---
  Est. Ref.: Adept Cobra s800 Base
  MoveJ (PreSustancia2)
  MoveJ (Sustancia2)

--- program PincharSustancia3 (robot myScara) ---
  Est. Ref.: Adept Cobra s800 Base
  MoveJ (PreSustancia3)
  MoveJ (Sustancia3)
  MoveJ (JeringaPreDown)

--- Python program MqttListener ---
import sys
sys.path.append(r"C:\RoboDK\Python")
sys.path.insert(0, r"C:\Users\algar\Desktop\PR2\PR2_RoboDK")

import paho.mqtt.client as mqtt
import importlib.util
import traceback
import threading


def cargar_modulo(nombre, ruta):
    spec = importlib.util.spec_from_file_location(nombre, ruta)
    modulo = importlib.util.module_from_spec(spec)
    spec.loader.exec_module(modulo)
    return modulo


robot_controller = cargar_modulo(
    "RobotController",
    r"C:\Users\algar\Desktop\PR2\PR2_RoboDK\RobotController.py"
)

scara_controller = cargar_modulo(
    "ScaraController",
    r"C:\Users\algar\Desktop\PR2\PR2_RoboDK\ScaraController.py"
)

print("RobotController cargado desde:", robot_controller.__file__)
print("ScaraController cargado desde:", scara_controller.__file__)


broker = "172.20.10.2"
puerto = 1883

station_commands_topic = "giirob/pr2/station/demo/commands"
station_status_topic = "giirob/pr2/station/demo/status"
temp_topic = "giirob/pr2/incubadora/temperatura"
scara_estado_topic = "scara/posiciones/estado"


def on_connect(client, userdata, flags, reason_code, properties=None):
    print("======================================")
    print("MQTT CONECTADO")
    print("Broker:", broker)
    print("Puerto:", puerto)
    print("Reason code:", reason_code)
    print("======================================")

    client.subscribe(station_commands_topic, 0)
    client.subscribe(temp_topic, 0)
    client.subscribe(scara_estado_topic, 0)

    print("Suscrito a:", station_commands_topic)
    print("Suscrito a:", temp_topic)
    print("Suscrito a:", scara_estado_topic)

    client.publish(station_status_topic, "listo")
    print("Publicado estado listo en:", station_status_topic)


def ejecutar_scara_en_hilo(mqttc, topic, payload):
    try:
        scara_controller.handle_message(mqttc, topic, payload)
    except Exception:
        print("ERROR en ScaraController:")
        traceback.print_exc()


def ejecutar_robot_en_hilo(mqttc, topic, payload):
    try:
        robot_controller.handle_message(mqttc, topic, payload)
    except Exception:
        print("ERROR en RobotController:")
        traceback.print_exc()


def on_message(mqttc, userdata, msg):
    topic = msg.topic.strip()
    payload = msg.payload.decode("utf-8").strip()

    print("\n======================================")
    print("MQTT LISTENER HA RECIBIDO MENSAJE")
    print("Topic:", topic)
    print("Payload:", payload)
    print("======================================")

    # --------------------------------------------------
    # MENSAJES DEL ESP32 PARA SCARA
    # --------------------------------------------------
    if topic == scara_estado_topic:
        print("Mensaje dirigido SOLO a ScaraController")

        try:
            scara_controller.handle_message(mqttc, topic, payload)
        except Exception:
            print("ERROR en ScaraController:")
            traceback.print_exc()

        return

    # --------------------------------------------------
    # MENSAJES DE TEMPERATURA PARA ROBOT CONTROLLER
    # --------------------------------------------------
    if topic == temp_topic:
        print("Mensaje dirigido SOLO a RobotController")

        try:
            robot_controller.handle_message(mqttc, topic, payload)
        except Exception:
            print("ERROR en RobotController:")
            traceback.print_exc()

        return

    # --------------------------------------------------
    # COMANDOS GENERALES
    # --------------------------------------------------
    if topic == station_commands_topic:
        comando = payload.lower().strip()

        if comando in [
            "start_gradilla",
            "start_scara",
            "star_gradiilla",
            "start_gradiilla"
        ]:
            print("Comando de gradilla dirigido SOLO a ScaraController EN HILO SEPARADO")

            hilo_scara = threading.Thread(
                target=ejecutar_scara_en_hilo,
                args=(mqttc, topic, payload),
                daemon=True
            )

            hilo_scara.start()
            return

        else:
            print("Comando dirigido SOLO a RobotController")

            hilo_robot = threading.Thread(
                target=ejecutar_robot_en_hilo,
                args=(mqttc, topic, payload),
                daemon=True
            )

            hilo_robot.start()
            return

    print("Topic no reconocido por MqttListener:", topic)


mqttc = mqtt.Client(mqtt.CallbackAPIVersion.VERSION2)
mqttc.on_connect = on_connect
mqttc.on_message = on_message

print("Conectando a MQTT...")
mqttc.connect(broker, puerto, 60)

print("MqttListener listo. Escuchando RobotController y ScaraController...")
mqttc.loop_forever()

--- Python program PresenciaSoporte ---
import sys
import time
import json
import math

# Ruta RoboDK
sys.path.append(r"C:\RoboDK\Python")

from robodk import robolink
from robodk.robomath import transl

import paho.mqtt.client as mqtt


# ============================================================
# CONFIGURACIÓN ROBO DK
# ============================================================

RDK = robolink.Robolink()

# Cambia este nombre si tu soporte se llama distinto en RoboDK
NOMBRE_SOPORTE = "Soporte1"

# Si tu objeto se llama Gradilla en vez de Soporte, cambia arriba por:
# NOMBRE_SOPORTE = "Gradilla"

# Sistema de referencia donde el operario deja la gradilla
NOMBRE_REFERENCIA_DEJADA = "Dejada"


# ============================================================
# CONFIGURACIÓN MQTT
# ============================================================

BROKER = "172.20.10.2"
PUERTO = 1883

TOPIC_COMANDOS = "giirob/pr2/station/demo/commands"

COMANDO_INICIO = "start_gradilla"

CLIENT_ID = "robodk_sensor_presencia_dejada"


# ============================================================
# CONFIGURACIÓN SENSOR VIRTUAL
# ============================================================

# Zona de detección dentro del sistema Dejada.
# Está en milímetros.
#
# Si el soporte está cerca del origen del sistema Dejada,
# se considera presente.
LIMITE_X_MM = 80
LIMITE_Y_MM = 80
LIMITE_Z_MM = 80

# Cada cuánto comprueba presencia
TIEMPO_ENTRE_LECTURAS = 0.5

# Para evitar mandar start_gradilla infinitas veces
comando_enviado = False


def obtener_item(nombre):
    item = RDK.Item(nombre)

    if not item.Valid():
        print("ERROR: No se encuentra en RoboDK:", nombre)
        return None

    print("OK encontrado en RoboDK:", nombre)
    return item


def conectar_mqtt():
    client = mqtt.Client(client_id=CLIENT_ID)

    print("Conectando a MQTT...")
    print("Broker:", BROKER)
    print("Puerto:", PUERTO)

    client.connect(BROKER, PUERTO, 60)
    client.loop_start()

    time.sleep(1)

    print("MQTT conectado")
    return client


def publicar_start_gradilla(mqttc):
    print("======================================")
    print("SOPORTE DETECTADO EN DEJADA")
    print("Enviando comando:", COMANDO_INICIO)
    print("Topic:", TOPIC_COMANDOS)
    print("======================================")

    mqttc.publish(TOPIC_COMANDOS, COMANDO_INICIO)


def obtener_posicion_relativa(objeto, referencia):
    """
    Devuelve x, y, z del objeto respecto al sistema de referencia Dejada.
    """

    pose_objeto_abs = objeto.PoseAbs()
    pose_ref_abs = referencia.PoseAbs()

    # Pose del objeto respecto al frame Dejada
    pose_relativa = pose_ref_abs.inv() * pose_objeto_abs

    x = pose_relativa.Pos()[0]
    y = pose_relativa.Pos()[1]
    z = pose_relativa.Pos()[2]

    return x, y, z


def soporte_esta_en_dejada(soporte, referencia):
    x, y, z = obtener_posicion_relativa(soporte, referencia)

    print("--------------------------------------")
    print("Posición soporte respecto a Dejada:")
    print("X:", round(x, 2), "mm")
    print("Y:", round(y, 2), "mm")
    print("Z:", round(z, 2), "mm")

    dentro_x = abs(x) <= LIMITE_X_MM
    dentro_y = abs(y) <= LIMITE_Y_MM
    dentro_z = abs(z) <= LIMITE_Z_MM

    if dentro_x and dentro_y and dentro_z:
        print("Resultado sensor: SOPORTE PRESENTE")
        return True
    else:
        print("Resultado sensor: no hay soporte")
        return False


def main():
    global comando_enviado

    print("======================================")
    print("SENSOR VIRTUAL DE PRESENCIA EN ROBO DK")
    print("======================================")

    soporte = obtener_item(NOMBRE_SOPORTE)
    referencia_dejada = obtener_item(NOMBRE_REFERENCIA_DEJADA)

    if soporte is None:
        print("Cambia NOMBRE_SOPORTE por el nombre real del objeto en RoboDK.")
        return

    if referencia_dejada is None:
        print("Cambia NOMBRE_REFERENCIA_DEJADA por el nombre real del frame en RoboDK.")
        return

    mqttc = conectar_mqtt()

    print("Sensor activo.")
    print("Esperando soporte en el sistema de referencia:", NOMBRE_REFERENCIA_DEJADA)

    while True:
        presente = soporte_esta_en_dejada(soporte, referencia_dejada)

        if presente and not comando_enviado:
            publicar_start_gradilla(mqttc)
            comando_enviado = True

        if not presente and comando_enviado:
            print("El soporte ha salido de Dejada. Sensor rearmado.")
            comando_enviado = False

        time.sleep(TIEMPO_ENTRE_LECTURAS)


if __name__ == "__main__":
    main()

--- Python program RobotController ---
import sys
sys.path.append(r"C:\RoboDK\Python")

from robodk import robolink
from robodk.robolink import ITEM_TYPE_ROBOT, ITEM_TYPE_TARGET
import time

RDK = robolink.Robolink()

# -----------------------------
# ROBOT / ROBO DK
# -----------------------------
ROBOT_NAME = "myRobotUR"

POS_SEGURA = "Incu2"
POS_PRE_INCUBADORA = "PrePlaceIncu"
POS_INCUBADORA = "PlaceIncu"

MECANISMO_INCUBADORA = "Refrigeradora"
DOOR_OPEN = "DoorOpen"
DOOR_CLOSE = "DoorClose"

# -----------------------------
# MQTT TOPICS
# -----------------------------
TOPIC_COMMANDS = "giirob/pr2/station/demo/commands"


def handle_message(mqttc, topic, payload):
    print("Topic recibido:", topic)
    print("Payload recibido:", payload)

    if topic != TOPIC_COMMANDS:
        print("Topic ignorado por RobotController:", topic)
        return

    comando = payload.strip().upper()

    if comando == "SACAR_GRADILLA":
        print("Orden recibida: SACAR_GRADILLA")
        proceso_sacar_gradilla()

    elif comando == "RESET":
        print("Reset recibido en RobotController")

    else:
        print("Comando no reconocido por RobotController:", comando)


def get_robot():
    robot = RDK.Item(ROBOT_NAME, ITEM_TYPE_ROBOT)

    if not robot.Valid():
        print("ERROR: robot no encontrado:", ROBOT_NAME)
        return None

    return robot


def get_target(nombre_target):
    target = RDK.Item(nombre_target, ITEM_TYPE_TARGET)

    if not target.Valid():
        print("ERROR: target no encontrado:", nombre_target)
        return None

    return target


def mover_robot(nombre_target):
    robot = get_robot()
    target = get_target(nombre_target)

    if robot is None or target is None:
        return False

    print("Moviendo robot a:", nombre_target)

    try:
        robot.MoveJ(target)
        robot.WaitMove()
        print("Robot llegó a:", nombre_target)
        return True

    except Exception as e:
        print("ERROR moviendo robot a", nombre_target, ":", e)
        return False


def mover_puerta(nombre_target):
    mecanismo = RDK.Item(MECANISMO_INCUBADORA)
    target = get_target(nombre_target)

    if not mecanismo.Valid():
        print("ERROR: mecanismo no encontrado:", MECANISMO_INCUBADORA)
        return False

    if target is None:
        return False

    print("Moviendo puerta a:", nombre_target)

    try:
        mecanismo.MoveJ(target)

        while mecanismo.Busy():
            time.sleep(0.1)

        print("Puerta movida a:", nombre_target)
        return True

    except Exception as e:
        print("ERROR moviendo puerta a", nombre_target, ":", e)
        return False


def ejecutar_programa(nombre_programa):
    print("\n======================================")
    print("Ejecutando programa:", nombre_programa)
    print("======================================")

    programa = RDK.Item(nombre_programa)

    if not programa.Valid():
        print("ERROR: no existe el programa:", nombre_programa)
        return False

    try:
        programa.RunProgram()

        while programa.Busy():
            time.sleep(0.1)

        time.sleep(0.2)

        print("Programa terminado:", nombre_programa)
        return True

    except Exception as e:
        print("ERROR ejecutando programa", nombre_programa, ":", e)
        return False


def coger_gradilla():
    print("\n======================================")
    print("COGIENDO GRADILLA / SOPORTE")
    print("======================================")

    if not ejecutar_programa("CerrarGarra"):
        return False

    if not ejecutar_programa("Adjuntar Soporte"):
        return False

    print("Gradilla/soporte cogido correctamente")
    return True


def ejecutar_lista_programas(programas):
    for nombre_programa in programas:
        ok = ejecutar_programa(nombre_programa)

        if not ok:
            print("Proceso detenido en:", nombre_programa)
            return False

    return True


def proceso_sacar_gradilla():
    print("\n======================================")
    print("INICIANDO PROCESO SACAR GRADILLA")
    print("======================================")

    # --------------------------------------------------
    # 1. Abrir incubadora
    # --------------------------------------------------
    if not mover_puerta(DOOR_OPEN):
        return

    time.sleep(1)

    # --------------------------------------------------
    # 2. Ir a la incubadora
    # --------------------------------------------------
    if not mover_robot(POS_PRE_INCUBADORA):
        return

    if not mover_robot(POS_INCUBADORA):
        return

    # --------------------------------------------------
    # 3. Coger soporte/gradilla
    # --------------------------------------------------
    if not coger_gradilla():
        return

    time.sleep(1)

    # --------------------------------------------------
    # 4. Sacar soporte de la incubadora
    # --------------------------------------------------
    if not mover_robot(POS_PRE_INCUBADORA):
        return

    if not mover_robot(POS_SEGURA):
        return

    # --------------------------------------------------
    # 5. Cerrar incubadora
    # --------------------------------------------------
    if not mover_puerta(DOOR_CLOSE):
        return

    print("Gradilla recogida correctamente")

    # --------------------------------------------------
    # 6. Ejecutar proceso posterior SIN SCARA
    # --------------------------------------------------
    programas_post_incubadora = [
        "DeIncuACentri",
        "MeterProbetas",
        "SacarProbetas",
        "DeCentriAPinchazo",
        "PrgramaAlchol",
        "DePinchazoACentri",
        "MeterProbetas",
        "SacarProbetas",
        "DeCentriARecogida",
        "HomeRobot",
        "ResetSoporte"
    ]

    ok = ejecutar_lista_programas(programas_post_incubadora)

    if not ok:
        return

    print("\n======================================")
    print("PROCESO COMPLETO TERMINADO CORRECTAMENTE")
    print("======================================")

--- Python program ScaraController ---
import json
import time
from robodk import robolink

RDK = robolink.Robolink()

# -----------------------------
# NOMBRES EN ROBODK
# -----------------------------
ROBOT_COLABORATIVO = "myRobotUR"
ROBOT_SCARA = "myScara"

PROGRAMA_INICIAL = "DeDejadaAPinchazo"

# IMPORTANTE:
# Crea estos 3 programas en RoboDK separando el antiguo Pinchar3Sustancias
PROGRAMA_SCARA_1 = "PincharSustancia1"
PROGRAMA_SCARA_2 = "PincharSustancia2"
PROGRAMA_SCARA_3 = "PincharSustancia3"

PROGRAMA_INCU = "DePinchazoAIncu"

MECANISMO_INCUBADORA = "Refrigeradora"

DOOR_OPEN = "DoorOpen"
DOOR_CLOSE = "DoorClose"

# -----------------------------
# TOPICS MQTT
# -----------------------------
TOPIC_COMANDOS = "giirob/pr2/station/demo/commands"
TOPIC_ORDEN_ESP32 = "scara/posiciones/respuestas"
TOPIC_ESTADO_ESP32 = "scara/posiciones/estado"
TOPIC_CONTROL_INCUBADORA = "giirob/pr2/incubadora/control"

# -----------------------------
# POSICIONES DE LA GRADILLA
# -----------------------------
posiciones = [
    "Pin1", "Pin2", "Pin3",
    "Pin4", "Pin5", "Pin6",
    "Pin7", "Pin8", "Pin9"
]

proceso_en_marcha = False
indice_actual = 0
mqttc_global = None


def obtener_item(nombre):
    item = RDK.Item(nombre)

    if not item.Valid():
        print("ERROR: No se encuentra en RoboDK:", nombre)
        return None

    print("OK encontrado en RoboDK:", nombre)
    return item


def detener_por_error():
    global proceso_en_marcha

    proceso_en_marcha = False

    print("======================================")
    print("PROCESO DETENIDO POR ERROR")
    print("======================================")


def ejecutar_programa(nombre_programa, esperar=True):
    print("\n======================================")
    print("Ejecutando programa:", nombre_programa)

    programa = obtener_item(nombre_programa)

    if programa is None:
        detener_por_error()
        return False

    programa.RunProgram()

    if esperar:
        programa.WaitFinished()

    print("Programa terminado:", nombre_programa)
    print("======================================")
    return True

def publicar_esp32(mensaje):
    global mqttc_global

    if mqttc_global is None:
        print("ERROR: mqttc_global es None. No puedo publicar al ESP32.")
        detener_por_error()
        return False

    payload = json.dumps(mensaje)

    print("Publicando al ESP32")
    print("Topic:", TOPIC_ORDEN_ESP32)
    print("Payload:", payload)

    try:
        info = mqttc_global.publish(TOPIC_ORDEN_ESP32, payload, qos=0)

        # Fuerza a que el publish se procese antes de seguir con RoboDK
        info.wait_for_publish(timeout=2)

        print("Mensaje MQTT enviado correctamente")
        return True

    except Exception as e:
        print("ERROR publicando al ESP32:", e)
        return False


def reset_leds_posicion(posicion):
    mensaje = {
        "posicion": posicion,
        "estado": "reset"
    }

    return publicar_esp32(mensaje)


def encender_led_sustancia(posicion, sustancia):
    mensaje = {
        "posicion": posicion,
        "estado": "inyectada",
        "sustancia": sustancia,
        "led": sustancia
    }

    return publicar_esp32(mensaje)

def ejecutar_scara_sincronizado(posicion):
    print("\n======================================")
    print("EJECUTANDO SCARA SINCRONIZADO")
    print("Posicion:", posicion)
    print("======================================")

    pasos = [
        (1, PROGRAMA_SCARA_1),
        (2, PROGRAMA_SCARA_2),
        (3, PROGRAMA_SCARA_3)
    ]

    for sustancia, programa in pasos:
        print("\n--------------------------------------")
        print("PREPARANDO SUSTANCIA", sustancia)
        print("Programa:", programa)
        print("--------------------------------------")

        # 1) Primero encendemos el LED de esa sustancia
        print("Encendiendo LED de sustancia", sustancia, "ANTES de inyectar")

        ok = encender_led_sustancia(posicion, sustancia)

        if not ok:
            print("ERROR encendiendo LED de sustancia:", sustancia)
            return False

        # Pequeña pausa para que el ESP32 tenga tiempo de encender el LED
        time.sleep(1.0)

        # 2) Ahora ejecutamos la inyección correspondiente
        print("Ejecutando inyección de sustancia", sustancia)

        ok = ejecutar_programa(programa, esperar=True)

        if not ok:
            print("ERROR ejecutando:", programa)
            return False

        print("Sustancia", sustancia, "inyectada correctamente")

        time.sleep(0.4)

    print("Las 3 sustancias han terminado en:", posicion)

    publicar_esp32({
        "posicion": posicion,
        "estado": "fin_posicion"
    })

    return True


def iniciar_proceso(mqttc):
    global proceso_en_marcha, indice_actual, mqttc_global

    if proceso_en_marcha:
        print("El proceso ya está en marcha. Ignoro nuevo comando.")
        return

    mqttc_global = mqttc
    proceso_en_marcha = True
    indice_actual = 0

    print("\n======================================")
    print("INICIANDO PROCESO COMPLETO DE GRADILLA")
    print("======================================")

    ok = ejecutar_programa(PROGRAMA_INICIAL, esperar=True)

    if not ok:
        detener_por_error()
        return

    mover_a_siguiente_posicion()


def mover_a_siguiente_posicion():
    global indice_actual, proceso_en_marcha

    if indice_actual >= len(posiciones):
        print("\n======================================")
        print("SE HAN PROCESADO LAS 9 POSICIONES")
        print("Ahora se mete la gradilla en la incubadora")
        print("======================================")

        ok = finalizar_gradilla_en_incubadora()

        if not ok:
            detener_por_error()
            return

        proceso_en_marcha = False

        print("\n======================================")
        print("PROCESO COMPLETO TERMINADO")
        print("Gradilla metida en la incubadora")
        print("Puerta cerrada")
        print("======================================")
        return

    posicion = posiciones[indice_actual]

    print("\n--------------------------------------")
    print("Moviendo robot colaborativo con MoveL a:", posicion)

    robot_ur = obtener_item(ROBOT_COLABORATIVO)
    target = obtener_item(posicion)

    if robot_ur is None or target is None:
        detener_por_error()
        return

    robot_ur.MoveL(target)
    robot_ur.WaitMove()

    print("Robot colaborativo ha llegado a:", posicion)

    # Apaga los 3 LEDs al comenzar cada pin.
    reset_leds_posicion(posicion)
    time.sleep(0.3)

    # Aquí se hace la nueva sincronización:
    # inyectar sustancia 1 -> LED 1
    # inyectar sustancia 2 -> LED 2
    # inyectar sustancia 3 -> LED 3
    ok = ejecutar_scara_sincronizado(posicion)

    if not ok:
        detener_por_error()
        return

    indice_actual += 1

    time.sleep(0.5)

    mover_a_siguiente_posicion()


def mover_puerta_incubadora(nombre_target):
    print("\n======================================")
    print("MOVIENDO PUERTA INCUBADORA A:", nombre_target)
    print("======================================")

    mecanismo = RDK.Item(MECANISMO_INCUBADORA)
    target = RDK.Item(nombre_target)

    if not mecanismo.Valid():
        print("ERROR: No se encuentra el mecanismo:", MECANISMO_INCUBADORA)
        return False

    if not target.Valid():
        print("ERROR: No se encuentra el target de puerta:", nombre_target)
        return False

    try:
        mecanismo.MoveJ(target)

        while mecanismo.Busy():
            time.sleep(0.1)

        print("Puerta movida correctamente a:", nombre_target)
        return True

    except Exception as e:
        print("ERROR moviendo puerta:", e)
        return False

def iniciar_lectura_temperatura_incubadora():
    global mqttc_global

    if mqttc_global is None:
        print("ERROR: mqttc_global es None. No puedo activar lectura temperatura.")
        return False

    mensaje = {
        "estado": "start_temp",
        "motivo": "soporte_dentro_puerta_cerrada"
    }

    payload = json.dumps(mensaje)

    print("\n======================================")
    print("ACTIVANDO LECTURA DE TEMPERATURA")
    print("Topic:", TOPIC_CONTROL_INCUBADORA)
    print("Payload:", payload)
    print("======================================")

    mqttc_global.publish(TOPIC_CONTROL_INCUBADORA, payload)
    return True

def finalizar_gradilla_en_incubadora():
    print("\n======================================")
    print("FASE FINAL: METER GRADILLA EN INCUBADORA")
    print("======================================")

    print("1) Abriendo puerta de la refrigeradora")
    ok = mover_puerta_incubadora(DOOR_OPEN)

    if not ok:
        print("ERROR abriendo puerta con target DoorOpen")
        return False

    time.sleep(0.5)

    print("2) Moviendo gradilla desde zona de pinchazo hasta incubadora")
    ok = ejecutar_programa(PROGRAMA_INCU, esperar=True)

    if not ok:
        print("ERROR ejecutando DePinchazoAIncu")
        return False

    time.sleep(0.5)

    print("3) Cerrando puerta de la refrigeradora")
    ok = mover_puerta_incubadora(DOOR_CLOSE)

    if not ok:
        print("ERROR cerrando puerta con target DoorClose")
        return False

    time.sleep(0.5)

    # Ahora sí: soporte dentro + puerta cerrada.
    # Activamos la lectura de temperatura en la ESP32.
    iniciar_lectura_temperatura_incubadora()

    print("FASE FINAL TERMINADA CORRECTAMENTE")
    return True

def procesar_estado_esp32(payload):
    try:
        data = json.loads(payload)
    except Exception as e:
        print("ERROR leyendo JSON del ESP32:", e)
        print("Payload recibido:", payload)
        return

    print("\n======================================")
    print("ESTADO RECIBIDO DEL ESP32")
    print("Payload:", data)
    print("======================================")

    posicion = str(data.get("posicion", "")).strip()
    estado = str(data.get("estado", "")).strip().lower()
    sustancia = data.get("sustancia", None)

    print("Posicion:", posicion)
    print("Estado:", estado)
    print("Sustancia:", sustancia)

def handle_message(mqttc, topic, payload):
    if isinstance(topic, bytes):
        topic = topic.decode("utf-8")

    if isinstance(payload, bytes):
        payload = payload.decode("utf-8")

    topic = topic.strip()
    payload = payload.strip()

    print("\n---- ScaraController recibe ----")
    print("Topic:", topic)
    print("Payload:", payload)
    print("--------------------------------")

    if topic == TOPIC_COMANDOS:
        comando = payload.lower().strip()

        if comando in [
            "start_gradilla",
            "start_scara",
            "star_gradiilla",
            "start_gradiilla"
        ]:
            iniciar_proceso(mqttc)

        else:
            print("Comando no reconocido para ScaraController:", comando)

        return

    if topic == TOPIC_ESTADO_ESP32:
        procesar_estado_esp32(payload)
        return

    print("Topic ignorado por ScaraController.")
